TEXTLIST HydraulicsConfigTabsTextList
  0 = 'General'
  1 = 'Top side - general'
  2 = 'Top side - pressure measurement'
  3 = 'Top side - frequency measurement'
  4 = 'Bottom side - general'
  5 = 'Bottom side - pressure measurement'
  6 = 'Bottom side - frequency measurement'
   = ''
END_TEXTLIST

(* stored: Version 1.1.0.1, ProductVersion 3.1.4018.5
   TextList HydraulicsConfigTabsTextList: Id {e9ef5449-58c2-42b0-b711-afb30c8d195b} *)
